# EPICS autosave request: EdwardsNextTurbo/EdwardsNextTurbo_settings.req
$(P):DISABLE
$(P):SET:NORMALSPEED
$(P):SET:STANDBYSPEED
